# EPICS autosave request: camera/simulator/autoSaveRestore/single_setting.req
# Cameras
file "camera_settings.req",	P=X2-CAM:
